# EPICS substitutions: evrSupport/Db/ioc/IOC-LR20-LS01pattern.substitutions
#
# Pattern records
file evrPatternAll.db {
#	    Device        ,  SLC Pattern Check LNK    , EVR/Trigger
#	                                                  Links
  pattern { DEVICE        ,        LINK4              , LINK5 , LINK6 }
	  { IOC:LR20:LS01 ,         ""                ,  ""   ,  ""   }
}
file evrEventAll.db {
  pattern { DEVICE }
	  { IOC:LR20:LS01}
}
